PROGRAM MAIN
VAR
END_VAR

Latch();
GVL.Number2:=GVL.Number1;
GVL.String1:='Hello';
GVL.Real1:=122222.566;

ACTION Latch:
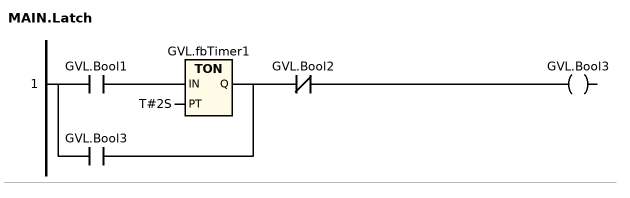
// NETWORK 1
GVL.fbTimer1(IN := GVL.Bool1, PT := T#2S); // TON
GVL.Bool3 := (GVL.fbTimer1.Q OR GVL.Bool3) AND NOT GVL.Bool2;
END_ACTION

END_PROGRAM

(* stored: Version 1.1.0.1, ProductVersion 3.1.4024.12
   POU MAIN: Id {de230d44-459a-4daf-b289-300bb0b126e0}, SpecialFunc None
   Action Latch: Id {66c0b85e-e85a-4677-98f5-aee2620f7c52} *)
